{attribute 'qualified_only'}
{attribute 'strict'}
TYPE eOperationMode :
(
	Auto := 0,
	Gridfollowing := 1,
	GridForming	:= 2
);
END_TYPE

(* stored: Version 1.1.0.1, ProductVersion 3.1.4026.18
   DUT eOperationMode: Id {d514c28d-fcbe-4c7f-83e8-f81e609adbc0} *)
